RoboDK station: kr10.rdk

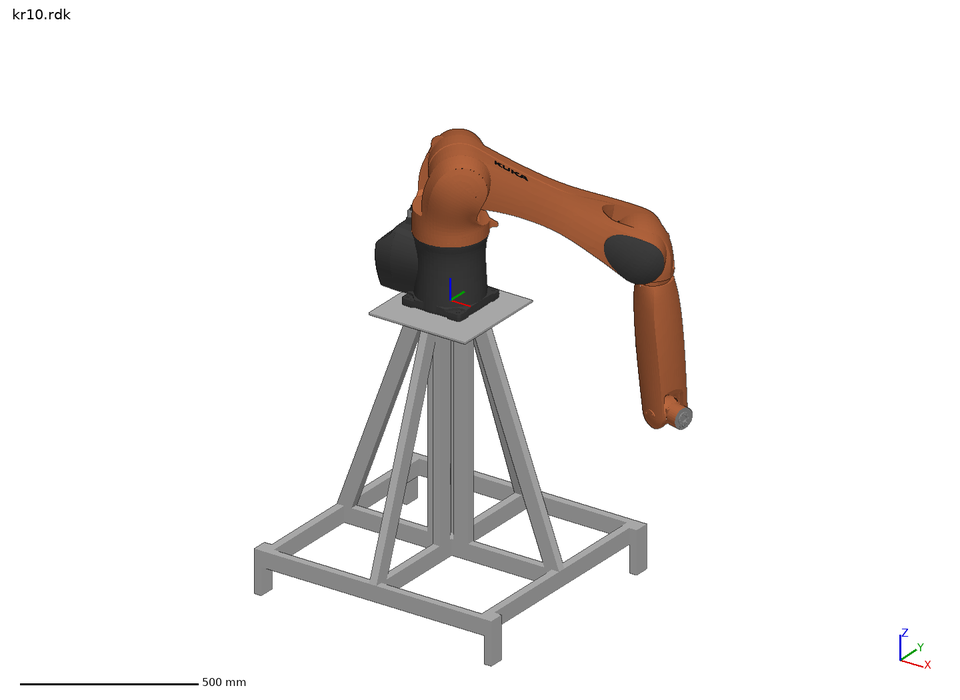
[picture v0: the station drawn from its stored meshes, robots at their saved joint values, targets as dots, program paths as lines]
Station kr10. Poses are relative to the parent item; angles as X-Y-Z fixed-axis rotations.
  - frame KUKA KR 10 R1100 sixx Base at (0, 0, 0) mm
    - robot KUKA KR 10 R1100 sixx: 6 axes, payload 10 kg, reach 1101 mm, repeatability 0.03 mm, weight 54 kg
        modified DH rows (alpha deg, a mm, theta deg, d mm): 0, 0, 0, 400; -90, 25, 0, 0; 0, 560, -90, 0; -90, 35, 0, 515; 90, 0, 0, 0; -90, 0, 180, 80
        joint limits [-110, -190, -120, -185, -120, -350] to [110, 45, 156, 185, 120, 350]; home [0, -90, 90, 0, 0, 0]; saved at [-37.342, 25.43, 60.405, 129.619, 85.755, -350]
  - object kuka base at (0, 0, 0) mm, size 812.8 x 762 x 857.2 mm, geometry from kuka base.stl
